// Mitsubishi GX Works2 project: FX2N   PLC: FX2N/FX2NC

PROGRAM MAIN
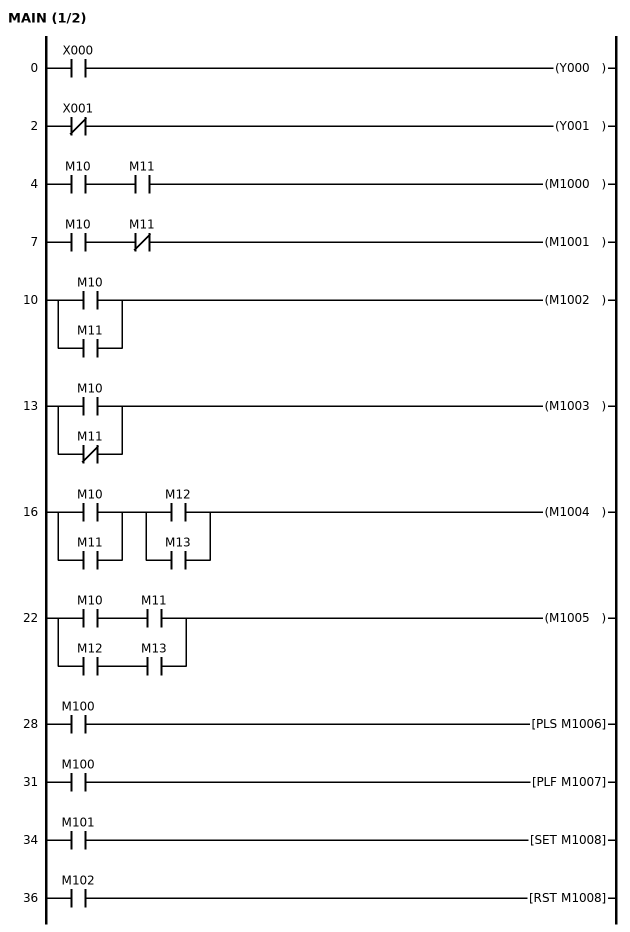
0     LD      X000
      OUT     Y000
2     LDI     X001
      OUT     Y001
4     LD      M10
      AND     M11
      OUT     M1000
7     LD      M10
      ANI     M11
      OUT     M1001
10    LD      M10
      OR      M11
      OUT     M1002
13    LD      M10
      ORI     M11
      OUT     M1003
16    LD      M10
      OR      M11
      LD      M12
      OR      M13
      ANB
      OUT     M1004
22    LD      M10
      AND     M11
      LD      M12
      AND     M13
      ORB
      OUT     M1005
28    LD      M100
      PLS     M1006
31    LD      M100
      PLF     M1007
34    LD      M101
      SET     M1008
36    LD      M102
      RST     M1008
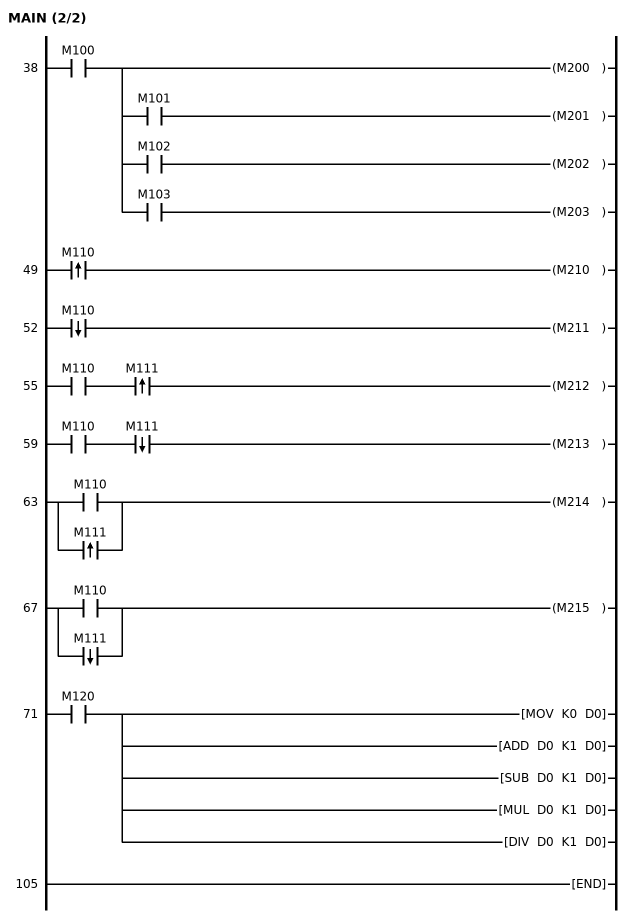
38    LD      M100
      OUT     M200
      MPS
      AND     M101
      OUT     M201
      MRD
      AND     M102
      OUT     M202
      MPP
      AND     M103
      OUT     M203
49    LDP     M110
      OUT     M210
52    LDF     M110
      OUT     M211
55    LD      M110
      ANDP    M111
      OUT     M212
59    LD      M110
      ANDF    M111
      OUT     M213
63    LD      M110
      ORP     M111
      OUT     M214
67    LD      M110
      ORF     M111
      OUT     M215
71    LD      M120
      MOV     K0 D0
      ADD     D0 K1 D0
      SUB     D0 K1 D0
      MUL     D0 K1 D0
      DIV     D0 K1 D0
105   END
END_PROGRAM
